FUNCTION_BLOCK DualModuleTmsSwitch IMPLEMENTS ITF_TmsSwitch
VAR_INPUT
	StateMachine : IPmlStateMachine;
END_VAR
VAR_OUTPUT
END_VAR
VAR
	_exchangeMover : IMover;
	_currentStation : ITF_SwitchStation;
	_demandPosition : MC_LREAL;
	_upPosition : MC_LREAL;
	_middlePosition : MC_LREAL;
	_downPosition : MC_LREAL;
	SwitchVelocity : MC_LREAL := 100.0;
	switchAxis : MC2_Axis_Base;
	arrTrackIds : ARRAY[1..4] OF OTCID := [16#010100F0,16#010100E0,16#010100D0,16#01010790];
	State :(
        Init,                                               
		Ready,                                 
        Enabling,
		Enabled,
		Resetting,
		Waiting,
		AssignMover,
		Moving,
		Done,
		Disabling); 
END_VAR

CASE State OF
	Init:
		IF NOT switchAxis.hasError() THEN
			State := Ready;
		END_IF
		
	Ready:
		IF StateMachine.GetCurrentState() = E_PMLState.ePMLState_Clearing THEN
			switchAxis.EnableAxis();
			State := Enabling;
		END_IF	
		
	Enabling:
		IF switchAxis.isEnabled() THEN
			State := Enabled;
		END_IF
		
	Enabled:
		IF StateMachine.GetCurrentState() = E_PMLState.ePMLState_Resetting THEN
			IF switchAxis.MoveTo(Position := _middlePosition, Velocity := 100.0) THEN
				State := Resetting;
			END_IF
		END_IF
		
	Resetting:
		IF switchAxis.isAtPosition(position := MiddlePosition) THEN
			State := Waiting;
		END_IF	
	
	Waiting:
		IF StateMachine.GetCurrentState() = E_PMLState.ePMLState_Aborting THEN
			switchAxis.DisableAxis();
			State := Disabling;
		END_IF
		
	AssignMover:
		IF HasMover() THEN
			IF FindNewTrack() <> 0 THEN
				State := Moving;
			END_IF
		ELSE
			State := Moving;
		END_IF

	Moving:	
		IF switchAxis.isAtPosition(_demandPosition) THEN
			State := Done;
		END_IF
	
	Done:
		IF _currentStation <> 0 THEN
			IF _currentStation.SwitchMoveComplete() THEN
				_exchangeMover := 0;
				_currentStation := 0;
			END_IF	
		END_IF
		State := Waiting;

	Disabling:
		IF NOT switchAxis.isEnabled() THEN
			State := Init;
		END_IF

END_CASE

switchAxis();

PROPERTY DownPosition : MC_LREAL
GET
DownPosition := _downPosition;
END_GET
SET
_downPosition := DownPosition;
END_SET
END_PROPERTY

METHOD PUBLIC ExchangeMover : BOOL
VAR_INPUT
	Mover : IMover;
	CurrentStation : ITF_SwitchStation;
END_VAR
IF _exchangeMover = 0 THEN
	_exchangeMover := Mover;	
	_currentStation := CurrentStation;
	ExchangeMover := TRUE;
END_IF
END_METHOD

METHOD PUBLIC FindNewTrack : OTCID
VAR_INPUT
END_VAR
VAR
	iTmsMover : ITmsMover;
END_VAR
IF __QUERYINTERFACE(_exchangeMover,iTmsMover) THEN
	IF Switch = SwitchState.Up THEN
		IF iTmsMover.ActiveTrack = arrTrackIds[3] THEN
			iTmsMover.ActivateTrack(newTrack := arrTrackIds[2]);
		END_IF
	ELSIF Switch = SwitchState.Middle THEN
		IF iTmsMover.ActiveTrack = arrTrackIds[1] THEN
			iTmsMover.ActivateTrack(newTrack := arrTrackIds[4]);
		ELSIF iTmsMover.ActiveTrack = arrTrackIds[2] THEN
			iTmsMover.ActivateTrack(newTrack := arrTrackIds[3]);
		END_IF
	ELSE
		IF iTmsMover.ActiveTrack = arrTrackIds[4] THEN
			iTmsMover.ActivateTrack(newTrack := arrTrackIds[1]);	
		END_IF
	END_IF
END_IF
FindNewTrack := iTmsMover.ActiveTrack;
END_METHOD

METHOD HasMover : BOOL
VAR_INPUT
END_VAR
HasMover := _exchangeMover <> 0;
END_METHOD

METHOD IsStationary : BOOL
VAR_INPUT
END_VAR
IsStationary := switchAxis.isStationary();
END_METHOD

PROPERTY PUBLIC MiddlePosition : MC_LREAL
GET
MiddlePosition := _middlePosition;
END_GET
SET
_middlePosition := MiddlePosition;
END_SET
END_PROPERTY

METHOD PUBLIC MoveTo : BOOL
VAR_INPUT
	positionState : SwitchState;
END_VAR
CASE positionState OF
	SwitchState.Down:
		IF NOT switchAxis.isAtPosition(position := _downPosition) THEN
			IF switchAxis.MoveTo(Position := _downPosition, Velocity := SwitchVelocity) THEN
				MoveTo := TRUE;
				State := AssignMover;
				_demandPosition := _downPosition;
			END_IF
		END_IF	
	SwitchState.Middle:
		IF NOT switchAxis.isAtPosition(position := _middlePosition) THEN
			IF switchAxis.MoveTo(Position := _middlePosition, Velocity := SwitchVelocity) THEN
				MoveTo := TRUE;
				State := AssignMover;
				_demandPosition := _middlePosition;
			END_IF
		END_IF	
	SwitchState.Up:
		IF NOT switchAxis.isAtPosition(position := _upPosition) THEN
			IF switchAxis.MoveTo(Position := _upPosition, Velocity := SwitchVelocity) THEN
				MoveTo := TRUE;
				State := AssignMover;
				_demandPosition := _upPosition;
			END_IF
		END_IF	
END_CASE
END_METHOD

PROPERTY PUBLIC Switch : SwitchState
GET
IF switchAxis.isAtPosition(position := _upPosition) THEN
	Switch := SwitchState.Up;
ELSIF switchAxis.isAtPosition(position := _middlePosition) THEN
	Switch := SwitchState.Middle;
ELSIF switchAxis.isAtPosition(position := _downPosition) THEN
	Switch := SwitchState.Down;
ELSE
	Switch := SwitchState.Moving;
END_IF
END_GET
END_PROPERTY

PROPERTY PUBLIC UpperPosition : MC_LREAL
GET
UpperPosition := _upPosition;
END_GET
SET
_upPosition := UpperPosition;
END_SET
END_PROPERTY

END_FUNCTION_BLOCK

(* stored: Version 1.1.0.1, ProductVersion 3.1.4024.11
   POU DualModuleTmsSwitch: Id {73ef316f-86b5-4cc1-962a-15251e072db1}, SpecialFunc None
   Property DownPosition: Id {513dbdb6-135b-46f3-8125-fc598ca8ce55}
   Get Get: Id {0db03243-0f6a-422c-b802-c5cc5c312e69}
   Set Set: Id {bbe8d847-123b-4a68-86bf-de9a0ef6b8f8}
   Method ExchangeMover: Id {b5f9d3d9-6f5f-4aaa-9562-32ebf7d41c8c}
   Method FindNewTrack: Id {64ec7bf3-c827-4335-99e4-b7418c5014bb}
   Method HasMover: Id {b10d08e7-730c-4533-8c1b-4e180c646997}
   Method IsStationary: Id {2f8bbf6e-5cce-4ab8-a9ba-43f43839d347}
   Property MiddlePosition: Id {a99e862a-0b65-4510-8ab1-7f0732d4e0cc}
   Get Get: Id {b34f701f-b631-47d2-ae36-146e9c98f154}
   Set Set: Id {9fbf98f9-449b-4537-a874-c25bab15bdec}
   Method MoveTo: Id {fd17c823-afe7-4820-9dad-912e69242e2b}
   Property Switch: Id {cea7677b-4e3e-436d-9a14-24ba96282e4e}
   Get Get: Id {955c8029-4c60-4733-8b6b-b2d2d74760a8}
   Property UpperPosition: Id {60deb3c6-3252-44f3-b5cb-16a8e597aa4b}
   Get Get: Id {f099d5c2-280a-458c-acd7-5c600c7a7194}
   Set Set: Id {bab004d1-8ed7-4888-a7ae-1210a1689e53} *)
